{attribute 'call_after_init'}
FUNCTION_BLOCK FB_MotionAxisDS402NC IMPLEMENTS I_MotionAxisDS402
VAR_INPUT
END_VAR
VAR_OUTPUT
END_VAR
VAR
    // perhaps use a structure no to repeat this code
    // derivation has a strong case here.
    iHome : I_HomeDS402;
    iHalt : I_Halt;
    iPower : I_Power;
    iReset : I_Reset;
    iMoveAbsolute : I_MoveAbsolute;
    iAxisParameters: I_AxisParameters;
    iAxisStatus : I_AxisStatus;
    iBacklashCompensation : I_BacklashCompensation;
    stDS402Drive : ST_DS402Drive;
    bError: BOOL;
    bBusy : BOOL;
    bDone : BOOL;
    bModeSet : BOOL;
    nErrorID: UDINT;
    sMessage : T_MAXSTRING;
    rtAbortDone : R_TRIG;
    rtDone : R_TRIG;
    nModeOfOperation : SINT;
    nModeOfOperationDisplay : SINT;
    bStartMove : BOOL;
    bOperational: BOOL;
END_VAR

(*Operation enbaled*)
IF stDS402Drive.stDriveStatus.ReadyToSwitchOn
    AND stDS402Drive.stDriveStatus.SwitchedOn
    AND stDS402Drive.stDriveStatus.OperationEnabled
    AND NOT stDS402Drive.stDriveStatus.Fault
    AND stDS402Drive.stDriveStatus.VoltageEnabled
    AND stDS402Drive.stDriveStatus.QuickStopActive
    AND NOT stDS402Drive.stDriveStatus.SwitchOnDisabled THEN
    bOperational := TRUE;
END_IF

// IF NOT bOperational THEN
//     //  Disclose loop operations
//     stDS402Drive.nDS402DriveControl:=16#0F;
// END_IF

// NB: Homing is stDS402Drive agnostice thus, these status must be passed cyclicly
// the status are hardware I/O provided, thus must be link to drive registers
THIS^.iHome.DS402Status(	ModeOfOperationDisplay:=THIS^.stDS402Drive.nModeOfOperationDisplay,
                            Bit13OpModeSpecific:=THIS^.stDS402Drive.stDriveStatus.Bit13_OpModeSpecific,
                            Bit12OpModeSpecific:=THIS^.stDS402Drive.stDriveStatus.Bit12_OpModeSpecific,
                            TargetReached:=THIS^.stDS402Drive.stDriveStatus.TargetReached );

// Homing routine must update the drive control and modeofoperation registers
IF THIS^.iHome.Busy THEN
    THIS^.stDS402Drive.nModeOfOperation := THIS^.iHome.DS402ModeOfOperation;
    THIS^.stDS402Drive.nDS402DriveControl:=THIS^.iHome.DS402Control;
END_IF

bBusy :=	THIS^.iHome.Busy;
bDone:=	THIS^.iHome.Done;
bError:=	THIS^.iHome.Error;
nErrorID:=	THIS^.iHome.ErrorID;

// Expose Axis Parameter
THIS^.iAxisParameters.ExposeAxisParams(Enable:=TRUE, RefreshDelay:=T#1S);
// Forward the abort event to homing block ( this is to sync the home state machine)
// Clear local execs flags after a completed move or a completed interruption
rtAbortDone(CLK:=(THIS^.iHalt.Done OR THIS^.iReset.Done));
IF  rtAbortDone.Q THEN
    THIS^.iMoveAbsolute.CommandMoveAbsolute := FALSE;
    THIS^.iHome.CommandMoveHome := FALSE;
    THIS^.bStartMove := FALSE;
    // forward global reset done event;

    THIS^.iHome.GlobalReset := THIS^.iReset.Done;
END_IF
// handle combined Errors conditions
THIS^.ErrorHandling();

PROPERTY AbortDone : BOOL
GET
AbortDone := THIS^.iHalt.Done OR THIS^.iReset.Done;
END_GET
END_PROPERTY

PROPERTY Aborted : BOOL
GET
ABorted := THIS^.iMoveAbsolute.Aborted;
END_GET
END_PROPERTY

METHOD AxisEnabled : BOOL
AxisEnabled:=THIS^.iAxisStatus.AxisEnabled();
END_METHOD

PROPERTY AxisParamsInit : BOOL
GET
AxisParamsInit := THIS^.iAxisParameters.AxisParamsInit;
END_GET
END_PROPERTY

PROPERTY AxisState : MC_AxisStates
GET
AxisState := THIS^.iAxisStatus.AxisState;
END_GET
END_PROPERTY

(*
    Handle positive/negative backlash compensation
    User needs to set the direction of backlash from the sign of the compensation value
    Backlash compensation is disabled during referencing (homing).
    When direction is positive/negative, further movement in the negative/positive direction not compensated
    further movement in the negative/positive direction will be compensated
*)
METHOD BacklashCompensation
VAR_INPUT
    Active     : BOOL;
    Compensation	: LREAL;
    RampVelocity	: LREAL;
    DisableMode	: E_DISABLEMODE := E_DISABLEMODE.DisableModeHold;
END_VAR
THIS^.iBacklashCompensation.BacklashCompensation(	Activate:=Active,
                                                    Compensation:=Compensation,
                                                    RampVelocity:=RampVelocity,
                                                    DisableMode:=DisableMode
                                                );
END_METHOD

(*synced Fbs need just to activate the compensation with a given ramp speed
  other parameters are provided via EPICS (declared in this FB) or via the more extended BackalshCompensation method (simulation) *)
METHOD BacklashCompensationActive
VAR_INPUT
    Active	: BOOL;
    RampVelocity	: LREAL;
END_VAR
THIS^.iBacklashCompensation.BacklashCompensationActive( Active:=Active,
                                                        RampVelocity:=RampVelocity );
END_METHOD

{warning 'Add property implementation'}
PROPERTY BacklashCompStatus : BOOL
GET
END_GET
END_PROPERTY

PROPERTY BacklashCompUserEn : BOOL
SET
THIS^.iBacklashCompensation.UserEnable:=BacklashCompUserEn;
END_SET
END_PROPERTY

PROPERTY Busy : BOOL
GET
Busy := THIS^.iHome.Busy OR THIS^.iMoveAbsolute.Busy;
END_GET
END_PROPERTY

PROPERTY Done : BOOL
GET
Done := THIS^.iHome.Done OR THIS^.iMoveAbsolute.Done;
END_GET
END_PROPERTY

PROPERTY Error : BOOL
GET
Error := bError;
END_GET
END_PROPERTY

METHOD ErrorHandling
(*
    Error from functions and Nc
    The error will send to EPICS interface based on predifined
    priority: axis, power, backlash, absoluteMove, etc...
*)
IF THIS^.iAxisStatus.Error  THEN
    bError:=THIS^.iAxisStatus.Error;
    nErrorId:=THIS^.iAxisStatus.ErrorID;
    sMessage := THIS^.iAxisStatus.Message;
ELSIF THIS^.iPower.Error AND THIS^.iPower.IsEnabled THEN
    bError:=THIS^.iPower.Error;
    nErrorId:=THIS^.iPower.ErrorID;
    sMessage := THIS^.iPower.Message;
ELSIF THIS^.iBacklashCompensation.Error THEN
    bError:=THIS^.iBacklashCompensation.Error;
    nErrorId:=THIS^.iBacklashCompensation.ErrorID;
    sMessage := THIS^.iBacklashCompensation.Message;
ELSIF THIS^.iMoveAbsolute.Error THEN
    bError:=THIS^.iMoveAbsolute.Error;
    nErrorId:=THIS^.iMoveAbsolute.ErrorID;
    sMessage := THIS^.iMoveAbsolute.Message;
ELSIF THIS^.iHome.Error (*Homing error*) THEN
    bError:=THIS^.iHome.Error;
    nErrorId:=THIS^.iHome.ErrorID;
    sMessage := THIS^.iHome.Message;
ELSIF THIS^.iHalt.Error AND THIS^.iHalt.Active THEN
    bError:=THIS^.iHalt.Error;
    nErrorId:=THIS^.iHalt.ErrorID;
    sMessage := THIS^.iHalt.Message;
ELSIF THIS^.iReset.Error  THEN
    bError:=THIS^.iReset.Error;
    nErrorId:=THIS^.iReset.ErrorID;
    sMessage := THIS^.iReset.Message;
ELSIF THIS^.iAxisParameters.Error THEN
    bError := THIS^.iAxisParameters.Error;
    nErrorId := THIS^.iAxisParameters.ErrorID;
    sMessage := THIS^.iAxisParameters.Message;
ELSE
    bError:=FALSE;
    nErrorId:=0;
    sMessage := '';
END_IF;
END_METHOD

PROPERTY ErrorID : UDINT
GET
ErrorID := THIS^.nErrorID;
END_GET
END_PROPERTY

METHOD ExposeAxisParams
VAR_INPUT
    Enable	: BOOL;
    RefreshDelay	: TIME;
END_VAR
THIS^.iAxisParameters.ExposeAxisParams(Enable:=Enable, RefreshDelay:=RefreshDelay);
END_METHOD

(*FB_Init is always available implicitly and it is used primarily for initialization.
The return value is not evaluated. For a specific influence, you can also declare the
methods explicitly and provide additional code there with the standard initialization
code. You can evaluate the return value.*)
METHOD FB_Init : BOOL
VAR_INPUT
    (* TRUE: the retain variables are initialized (reset warm / reset cold)*)
    bInitRetains	: BOOL;
    (* TRUE: the instance will be copied to the copy code afterward (online change)*)
    bInCopyCode	: BOOL;
    iHome : I_HomeDS402;
    iHalt : I_Halt;
    iPower : I_Power;
    iReset : I_Reset;
    iMoveAbsolute : I_MoveAbsolute;
    iAxisParameters: I_AxisParameters;
    iAxisStatus : I_AxisStatus;
    iBacklashCompensation : I_BacklashCompensation;
END_VAR
THIS^.iHome := iHome;
THIS^.iHalt := iHalt;
THIS^.iPower := iPower;
THIS^.iReset := iReset;
THIS^.iMoveAbsolute := iMoveAbsolute;
THIS^.iAxisParameters:= iAxisParameters;
THIS^.iAxisStatus := iAxisStatus;
THIS^.iBacklashCompensation  := iBacklashCompensation ;
END_METHOD

METHOD Halt
VAR_INPUT
    Execute	: BOOL;
    Deceleration	: LREAL := 0;
    Jerk	: LREAL := 0;
    BufferMode	: MC_BufferMode := MC_BufferMode.MC_Aborting;
END_VAR
THIS^.iHalt.Halt( Execute:=Execute,
                     Deceleration:=Deceleration,
                    Jerk:=Jerk ,
                    BufferMode:=BufferMode );
END_METHOD

{warning 'Add property implementation'}
PROPERTY HaltActive : BOOL
GET
END_GET
END_PROPERTY

{warning 'Add property implementation'}
PROPERTY HaltBusy : BOOL
GET
END_GET
END_PROPERTY

PROPERTY HaltDone : BOOL
GET
HaltDone := THIS^.iHalt.Done;
END_GET
END_PROPERTY

METHOD Home
VAR_INPUT
    Execute	: BOOL;
    HomeSpeedFast	: LREAL;
    HomeSpeedSlow	: LREAL;
END_VAR
// then call the
THIS^.iHome.Home(Execute:=Execute, HomeSpeedFast:=HomeSpeedFast, HomeSpeedSlow:=HomeSpeedSlow);
END_METHOD

PROPERTY HomeBusy : BOOL
GET
HomeBusy := THIS^.iHome.Busy;
END_GET
END_PROPERTY

PROPERTY HomeDone : BOOL
GET
HomeDone := THIS^.iHome.Done;
END_GET
END_PROPERTY

{warning 'Add property implementation'}
PROPERTY HomeMode : E_EpicsHomeCmd
GET
HomeMode := THIS^.iHome.Mode;
END_GET
END_PROPERTY

PROPERTY InTargetPosition : BOOL
GET
InTargetPosition := THIS^.iAxisStatus.InTargetPosition;
END_GET
END_PROPERTY

PROPERTY MeasuredAcceleration : LREAL
GET
MeasuredAcceleration := THIS^.iAxisStatus.MeasuredAcceleration;
END_GET
END_PROPERTY

PROPERTY MeasuredCompensation : LREAL
GET
MeasuredCompensation := THIS^.iBacklashCompensation.ActCompensation;
END_GET
END_PROPERTY

PROPERTY MeasuredPosition : LREAL
GET
MeasuredPosition := THIS^.iAxisStatus.MeasuredPosition;
END_GET
END_PROPERTY

PROPERTY MeasuredPositionDiff : LREAL
GET
MeasuredPositionDiff := THIS^.iAxisStatus.MeasuredPositionDiff;
END_GET
END_PROPERTY

PROPERTY MeasuredVelocity : LREAL
GET
MeasuredVelocity := THIS^.iAxisStatus.MeasuredVelocity;
END_GET
END_PROPERTY

PROPERTY Message : T_MaxString
GET
Message :=sMessage;
END_GET
END_PROPERTY

METHOD ModeOfOperation : BOOL;
VAR_INPUT
    RecentModeOfOperation : E_DS402OpMode;
END_VAR
THIS^.bModeSet := FALSE;
IF THIS^.stDS402Drive.nModeOfOperationDisplay <> RecentModeOfOperation THEN
    THIS^.stDS402Drive.nModeOfOperation := RecentModeOfOperation;
    THIS^.bModeSet := FALSE;
ELSE
    THIS^.bModeSet := TRUE;
END_IF

ModeOfOperation := THIS^.bModeSet;
END_METHOD

METHOD MoveAbsolute
VAR_INPUT
    Execute     : BOOL;
    Position	: LREAL;
    Velocity	: LREAL;
    Acceleration	: LREAL := 0.0;
    Deceleration	: LREAL := 0.0;
    Jerk	: LREAL := 0.0;
    BufferMode	: MC_BufferMode := MC_BufferMode.MC_Aborting;
END_VAR
THIS^.iMoveAbsolute.MoveAbsolute( 	Execute:=Execute,
                                    Position:=Position,
                                       Velocity := Velocity,
                                    Acceleration := Acceleration,
                                    Deceleration := Deceleration,
                                    Jerk := Jerk,
                                    BufferMode := BufferMode);
END_METHOD

{warning 'Add property implementation'}
PROPERTY MoveAbsoluteAborted : BOOL
GET
MoveAbsoluteAborted := THIS^.iMoveAbsolute.Aborted;
END_GET
END_PROPERTY

{warning 'Add property implementation'}
PROPERTY MoveAbsoluteActive : BOOL
GET
END_GET
END_PROPERTY

PROPERTY MoveAbsoluteBusy : BOOL
GET
MoveAbsoluteBusy := THIS^.iMoveAbsolute.Busy;
END_GET
END_PROPERTY

{warning 'Add property implementation'}
PROPERTY MoveAbsoluteDone : BOOL
GET
MoveAbsoluteDone := THIS^.iMoveAbsolute.Done;
END_GET
END_PROPERTY

PROPERTY NegativeMotionIsEnabled : BOOL
GET
 NegativeMotionIsEnabled := THIS^.iAxisStatus.NegativeMotionIsEnabled;
END_GET
END_PROPERTY

PROPERTY PositiveMotionIsEnabled : BOOL
GET
PositiveMotionIsEnabled := THIS^.iAxisStatus.PositiveMotionIsEnabled;
END_GET
END_PROPERTY

METHOD Power
VAR_INPUT
    Enable	: BOOL;
    Enable_Positive	: BOOL;
    Enable_Negative	: BOOL;
    Override	: LREAL := 100.0;
    BufferMode	: MC_BufferMode := MC_BufferMode.MC_Aborting;
END_VAR
THIS^.iPower.Power(	Enable:=Enable,
                    Enable_Positive:= Enable_Positive,
                    Enable_Negative:=Enable_Negative,
                    Override:=Override,
                    BufferMode:=BufferMode
                );
END_METHOD

{warning 'Add property implementation'}
PROPERTY PowerActive : BOOL
GET
END_GET
END_PROPERTY

(*This is overriden by this object internal acess to the interlock instance
  this is intended to pass power enable flags via the fbMotionDrive
*)
METHOD PowerEnables
VAR_INPUT
    Enable	: BOOL;
    Enable_Positive	: BOOL;
    Enable_Negative	: BOOL;
END_VAR
THIS^.iPower.Power(	Enable:=Enable,
                    Enable_Positive:= Enable_Positive,
                    Enable_Negative:=Enable_Negative,
                    Override:=100.0,
                    BufferMode:=MC_BufferMode.MC_Aborting
                );
END_METHOD

PROPERTY PowerIsEnabled : BOOL
GET
END_GET
END_PROPERTY

{warning 'Add property implementation'}
PROPERTY PowerOverride : LREAL
GET
PowerOverride := THIS^.iPower.Override;
END_GET
END_PROPERTY

METHOD Reset
VAR_INPUT
    Execute	: BOOL;
END_VAR
THIS^.iReset.Reset(Execute:=Execute);
END_METHOD

PROPERTY ResetBusy : BOOL
GET
ResetBusy := THIS^.iReset.Busy;
END_GET
END_PROPERTY

PROPERTY ResetDone : BOOL
GET
ResetDone := THIS^.iReset.Done;
END_GET
END_PROPERTY

PROPERTY RestoreDone : BOOL
GET
RestoreDone := THIS^.iAxisParameters.RestoreDone;
END_GET
END_PROPERTY

PROPERTY SavedPosition : LREAL
GET
SavedPosition := THIS^.iAxisParameters.SavedPosition;
END_GET
END_PROPERTY

PROPERTY ScaledEncoderCount : UDINT
GET
ScaledEncoderCount := THIS^.iAxisParameters.ScaledEncoderCount;
END_GET
END_PROPERTY

{warning 'Add property implementation'}
PROPERTY StandStill : BOOL
GET
StandStill := THIS^.iAxisStatus.StandStill;
END_GET
END_PROPERTY

(*
    Check all post condition before updating bCommandedMoveAbsolute
    The implmentatation will depend on the axis type
    DS402 NC/Direct axis : Implementation need to check that the drive is in the correct mode before initaiting the move then set bCommandedMoveAbsolute
    MP NC axis : will immediately write to bCommandedMoveAbsolute
*)
METHOD StartMove : BOOL
VAR_INPUT
    MoveMode	: E_EpicsMotorCmd;
    CmdExecute	: BOOL;
END_VAR
THIS^.bStartMove := FALSE;
CASE MoveMode  OF
    E_EpicsMotorCmd.MOVE_ABSOLUTE:
        IF THIS^.ModeOfOperation(RecentModeOfOperation:=8) THEN
            THIS^.iMoveAbsolute.CommandMoveAbsolute := CmdExecute AND bOperational;
            THIS^.bStartMove := TRUE;
        END_IF

    E_EpicsMotorCmd.HOME:
        IF THIS^.ModeOfOperation(RecentModeOfOperation:=6) THEN
            THIS^.iHome.Home( Execute:=CmdExecute AND bOperational,
                                HomeSpeedFast:=THIS^.iAxisParameters.RefVeloSearch,
                                HomeSpeedSlow:=THIS^.iAxisParameters.RefVeloSync );
            THIS^.bStartMove := TRUE;
        END_IF

END_CASE
// for typical NC axis no further tests needed
StartMove := THIS^.bStartMove;
END_METHOD

PROPERTY Stopped : BOOL
GET
Stopped := THIS^.iAxisStatus.Stopped;
END_GET
END_PROPERTY

END_FUNCTION_BLOCK

(* stored: Version 1.1.0.1
   POU FB_MotionAxisDS402NC: Id {0e4f30c7-9701-46fd-b9a3-891c9877e9a0}, SpecialFunc None
   Property AbortDone: Id {374c53b8-e916-472e-ade8-b85325191589}
   Get Get: Id {6b245bad-f401-4f8e-9264-4a2584d556cc}
   Property Aborted: Id {4156e934-1b40-4455-a852-d13a6f85e247}
   Get Get: Id {f64d8356-b5c6-48bb-b87b-e3ae7c0b7754}
   Method AxisEnabled: Id {ca10feff-4ca4-4f00-8af9-2ad21dbd4fe1}
   Property AxisParamsInit: Id {32334eb8-10f2-4d07-ab5b-86ebcd5e11a9}
   Get Get: Id {c98ae9f4-6b0e-43dd-855d-ea9149414625}
   Property AxisState: Id {9181aaf9-63c5-483a-98c8-6f4d56052b84}
   Get Get: Id {762e0479-bef5-4ed2-8a61-2fa227a0fbc7}
   Method BacklashCompensation: Id {3cbfe54b-fca5-4a08-b7dd-54501e2befa1}
   Method BacklashCompensationActive: Id {4d3c7c36-fb90-4b0f-9a3e-ed6c33ee0af5}
   Property BacklashCompStatus: Id {f644499f-f560-492d-91c8-383f5866b106}
   Get Get: Id {b03b55e8-e4d2-411d-a256-be8f86227bd3}
   Property BacklashCompUserEn: Id {e14ee1fc-526a-41de-bf16-0f34a34b5dd8}
   Set Set: Id {9ff60291-485b-49f5-8d73-ff6ca3f74134}
   Property Busy: Id {578b3c05-4979-42ec-a4d0-8e76f72dc0fa}
   Get Get: Id {e6e5c3cc-a354-4dce-8e29-2956aae35a29}
   Property Done: Id {981479f9-c694-4d1a-be9a-1752e6deb595}
   Get Get: Id {91103579-069e-4364-b8aa-ad07e400a647}
   Property Error: Id {9fe1588b-412f-4605-918b-c5f99c799aa8}
   Get Get: Id {c4e6bfd0-9a24-4e18-b425-f001b24ab2c0}
   Method ErrorHandling: Id {343e873e-1fe5-4eb8-99b8-88802101a3d0}
   Property ErrorID: Id {62fe70e2-cbbe-4206-8465-ac97709764ea}
   Get Get: Id {adeaeec9-70c6-46d4-8459-1ae1d32f2798}
   Method ExposeAxisParams: Id {a632f118-6207-4571-87e6-5c8ea26bb9ec}
   Method FB_Init: Id {1dac3e04-3581-442d-91f0-9c2dc1b453ee}
   Method Halt: Id {d4ec37ef-180a-4be0-827e-94d1034c9fea}
   Property HaltActive: Id {35227419-4529-4956-aa2d-48519159746f}
   Get Get: Id {0d2c6a63-e105-4274-9270-84e6cefd82f6}
   Property HaltBusy: Id {93f9fecf-b17d-42c9-a5c3-52833b5d3ce2}
   Get Get: Id {fdfff023-0454-434e-94aa-756ad214aada}
   Property HaltDone: Id {86288e35-2305-4f09-b91e-62b5f3ac95b1}
   Get Get: Id {748043de-3db2-4500-91f8-17ae79bb0d56}
   Method Home: Id {eb6ca2c3-dadc-488d-aa64-29befcb2a8c6}
   Property HomeBusy: Id {120358f8-1638-4a9d-846b-d914e71b3608}
   Get Get: Id {d96b7d9f-05a4-416a-b556-429a717df190}
   Property HomeDone: Id {546d39e6-f883-4c11-9aab-5aa9ff4d09c0}
   Get Get: Id {4a3157da-152a-443d-9f98-241770a79ad1}
   Property HomeMode: Id {b93e43bf-64d4-49dd-914c-3ebb62170b14}
   Get Get: Id {622801fe-c552-45ac-a4f2-6aeabaf9494b}
   Property InTargetPosition: Id {4d445891-163f-4111-83eb-60f09ddee9d3}
   Get Get: Id {78eb0d62-9d11-498f-9b62-d0ea3022166c}
   Property MeasuredAcceleration: Id {fde439bd-ceac-447d-b568-038bedb4787b}
   Get Get: Id {6817404e-1f00-4263-9e20-e124994469e2}
   Property MeasuredCompensation: Id {2e022ece-f4bb-4740-bf80-f212d43fd71f}
   Get Get: Id {51a19da8-1a6e-4644-9321-5c1f9eef648e}
   Property MeasuredPosition: Id {6cf29060-4b4f-441e-be73-6bd263e8a5e1}
   Get Get: Id {ece6ca55-4e88-4e0c-90de-6b353d74e67c}
   Property MeasuredPositionDiff: Id {0218e957-e0a4-4da4-976c-945e9f411fbc}
   Get Get: Id {90598c1b-8361-437f-b77f-7a6dad08ddaf}
   Property MeasuredVelocity: Id {6b852a66-e760-4085-88e2-79922e5f7ea6}
   Get Get: Id {62e95f94-4579-4306-a03b-7cf42338fcc9}
   Property Message: Id {beedbba4-7ec8-43f2-bdf8-e3dfd5016351}
   Get Get: Id {97f605d0-b60f-4441-9824-809353c47817}
   Method ModeOfOperation: Id {b52ebe5d-9983-420e-838a-c6d4f4dd39c1}
   Method MoveAbsolute: Id {781fcd7e-4774-4268-81a1-b3c3c7f5e72f}
   Property MoveAbsoluteAborted: Id {5813dcd7-b1f8-48f9-9b13-3719479eeba2}
   Get Get: Id {98863092-2796-4164-90ef-b53e25045c41}
   Property MoveAbsoluteActive: Id {373314df-6b0c-466e-b451-6706f56ed883}
   Get Get: Id {387115e3-2e0c-4c0c-99bd-7616b9c161ed}
   Property MoveAbsoluteBusy: Id {90de2003-6a05-43e8-a6c2-96aedbe6d620}
   Get Get: Id {1daf24c7-87ab-4eff-899e-03b4a03ab146}
   Property MoveAbsoluteDone: Id {8f337d45-ab01-4450-b8b4-8d2bd030948b}
   Get Get: Id {f717b2f3-066e-4bce-bc8a-19c7bb7803ed}
   Property NegativeMotionIsEnabled: Id {3c58869b-58ac-4c04-944f-b7005522293b}
   Get Get: Id {25ade829-9743-4ef2-9ada-5abe4c62fcf0}
   Property PositiveMotionIsEnabled: Id {756ccefa-9794-406c-b18f-ed07b52748cb}
   Get Get: Id {c952e9da-eba6-43bb-abc2-d1df33626a0f}
   Method Power: Id {fc0aa584-ea73-4eaf-8938-15ff0a2d5f6a}
   Property PowerActive: Id {376b2784-c771-437d-972f-22133de5b9be}
   Get Get: Id {5a504d25-7794-45ea-926d-8dcb2e39688b}
   Method PowerEnables: Id {97836c2c-1367-4cdd-a741-88828ffd0436}
   Property PowerIsEnabled: Id {2019a017-227c-47b7-97fb-dff4903aafb2}
   Get Get: Id {22a4346b-0f2c-469d-a930-057b483384d8}
   Property PowerOverride: Id {664d80c1-5f23-4e82-a16f-5bce8a03ec15}
   Get Get: Id {e02576f5-9fac-4947-a087-f064c2825885}
   Method Reset: Id {4d4369f8-943f-4a1c-a1c1-d8b2bbc9be87}
   Property ResetBusy: Id {d88f6672-c5e1-43f0-ab40-95f72b3ff1a4}
   Get Get: Id {172077a0-36c2-4fa0-bd0b-e832b74f5cbf}
   Property ResetDone: Id {b2e117ae-ea92-4c10-8a70-709b9a0506f1}
   Get Get: Id {1453bf42-1fdf-4ef2-9e87-ead3dabc873f}
   Property RestoreDone: Id {735ea9de-27f6-4b5a-915f-5995f7f868c7}
   Get Get: Id {fbd606c9-1af0-4c90-ba85-1e171c0c87a5}
   Property SavedPosition: Id {aa926740-9773-4290-acbd-1ab4f19e25fa}
   Get Get: Id {50656452-8223-45aa-909c-1b7b5589f360}
   Property ScaledEncoderCount: Id {cfa53524-89d7-4373-b39a-6d14131d0381}
   Get Get: Id {65b107b5-f09c-47a5-ba19-4140d478c782}
   Property StandStill: Id {9c4fc74f-cbef-4500-bc30-6594fe99030f}
   Get Get: Id {dfbc2698-2c48-4be9-adc8-c7a6e9db2cd8}
   Method StartMove: Id {ae3a68ed-e6ae-4591-9660-a38d4c1bbcc8}
   Property Stopped: Id {3fc8dd04-b557-4a21-8f7b-99bb919123a1}
   Get Get: Id {eaab0962-a193-4b99-98ea-dcdb5bfcef43} *)
